// TIA Portal V16 export
// export: Created 2023-03-29T11:03:45.0564835Z, ExportSetting WithDefaults, DisplayName Totally Integrated Automation Portal, DisplayVersion V16 Update 6, DisplayName TIA Portal Version Control Interface, DisplayVersion V16 Update 2, DisplayName TIA Portal Openness, DisplayVersion V16 Update 6, DisplayName STEP 7 Professional, DisplayVersion V16 Update 6, DisplayName STEP 7 Safety, DisplayVersion V16, DisplayName WinCC Advanced, DisplayVersion V16 Update 6
VAR_GLOBAL   // PLC tag table "Z6"
   inputAumagotowośćZ_6 AT %M65.0 : Bool;   // znacznik wejście
   Hbit_Reset_Z6 AT %M20.6 : Bool;
   Hbit_Zamknij_Z6 AT %M20.5 : Bool;
   inputAumaautomatZ_6 AT %M64.7 : Bool;   // znacznik wejście
   setSVMO_Z_6 AT %M65.2 : Bool;   // Znacznik polecenia otwórz w trybie automat
   inputAumalokalneZ_6 AT %M64.6 : Bool;   // znacznik wejście
   Hbit_Auto_Manu_Z6 AT %M20.7 : Bool;
   inputREMT_Z_6 AT %M64.1 : Bool;   // znacznik wejście zdalne
   inputAwariaMomentZ_6 AT %M64.5 : Bool;   // znacznik wejście
   Hbit_Otwórz_Z6 AT %M20.4 : Bool;
   isAUMA_Z_6 AT %M52.7 : Bool;   // przęłącznik wymiany na AUMA
   Hbit_REN_Z6 AT %M20.2 : Bool;
   CMD_Open_Z_6 AT %M65.5 : Bool;   // załącz otwieranie
   Hbit_Alarm_Z6 AT %M20.0 : Bool;
   Hbit_Otwarta_Z6 AT %M20.1 : Bool;
   CMD_Awaria_Z_6 AT %M65.7 : Bool;   // Awaria zbiorcza
   Hbit_Zamknieta_Z6 AT %M20.3 : Bool;
   CMD_Close_Z_6 AT %M65.6 : Bool;   // załącz zamykanie
   inputRuch_Z_6 AT %M64.4 : Bool;
   setSVMC_Z_6 AT %M65.3 : Bool;   // Znacznik polecenia zamknij w trybie automat
   isGotowość_Z_6 AT %M64.0 : Bool;   // bit gotowości wspólny
   Byte_Status_Z6 AT %MW20 : Word;   // Słowo statusu napędu
   setAlarm_Moment_Z_6 AT %M65.4 : Bool;   // znacznik alarmu od momentówki w trybie zdalnym (aut/mamnual)
   inputZamkniętaZ_6 AT %M64.3 : Bool;   // znacznik wejście
   inputOtwartaZ_6 AT %M64.2 : Bool;   // znacznik wejście
   inputAumaawariaZ_6 AT %M65.1 : Bool;   // znacznik wejście
   edge_Hz_Z6 AT %M92.2 : Bool;   // pamięć zbocza 1 Hz
END_VAR
